(* PLC project ap_master2, Dassault Systèmes ControlBuild 2024x Refresh1 *)
(* stored: creationDateTime 2024-04-12T15:40:51-01:00 *)

PROGRAM ap_master2.ap_master2

(* FBD diagram, written out as Structured Text *)
END_PROGRAM
